# EPICS autosave request: apps/vmeCratesApp/Db/vmeGroupSettings.req
$(GROUP)t_set
$(GROUP)man_set
$(GROUP)cpid_loc_mod
$(GROUP)cpid_man_mod
$(GROUP)cpid_dsbl
$(GROUP)cpid_kp
$(GROUP)cpid_ki
$(GROUP)cpid_kd
